PROGRAM Arbeitsplan
VAR
	Schritt_1		:Skill_1;
	Schritt_2		:Sequenz_1;
	
	Check			:BOOL;
	
	Var_1			:BOOL;
	Var_2			:BOOL;
	Var_3			:BOOL;
	Var_4			:BOOL;
END_VAR

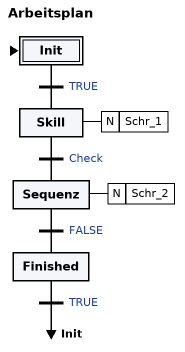
INITIAL_STEP Init:
END_STEP
TRANSITION FROM Init TO Skill
    := TRUE;
END_TRANSITION
STEP Skill:
    Schr_1(N);
END_STEP
TRANSITION FROM Skill TO Sequenz
    := Check;
END_TRANSITION
STEP Sequenz:
    Schr_2(N);
END_STEP
TRANSITION FROM Sequenz TO Finished
    := FALSE;
END_TRANSITION
STEP Finished:
END_STEP
TRANSITION FROM Finished TO Init
    := TRUE;
END_TRANSITION

ACTION Schr_1:
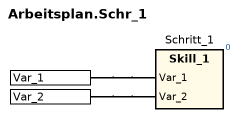
Schritt_1(Var_1 := Var_1, Var_2 := Var_2); // Skill_1
END_ACTION

ACTION Schr_2:
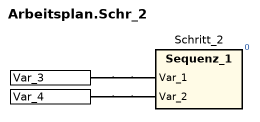
Schritt_2(Var_1 := Var_3, Var_2 := Var_4); // Sequenz_1
END_ACTION

END_PROGRAM

(* stored: Version 1.1.0.1
   POU Arbeitsplan: Id {19c96af4-f292-4baa-98e6-42cbe8df2e92}, SpecialFunc None
   Action Schr_1: Id {6747d966-225f-4188-96db-890c56409d1f}
   Action Schr_2: Id {2608489b-19c0-4532-8e23-23cf451e0273} *)
